TYPE ST_RecipeData :
STRUCT
	Receipt1 : INT;
	Receipt2 : INT;
END_STRUCT
END_TYPE

(* stored: Version 1.1.0.1, ProductVersion 3.1.4018.2
   DUT ST_RecipeData: Id {f7f700d3-277f-4478-b4eb-a2531fd01af1} *)
